(* PLC project contactor_1dir_2speed, Dassault Systèmes ControlBuild 2024x *)
(* stored: creationDateTime 2023-10-03T11:13:14-01:00 *)

(* This module simulates control system of motor. This motor has one direction and two speeds. This system is represented by two contactors. *)
FUNCTION_BLOCK equipment_library.contactor_1dir_2speed
  VAR_INPUT
    voltage380 : BOOL := true;
    cmdSupply : BOOL := true;
    sensorSupply : BOOL := true;
  END_VAR
  VAR_INPUT
    highSpeed : BOOL := false;
    lowSpeed : BOOL := false;
  END_VAR
  VAR_OUTPUT
    fwdHsState : BOOL := false;
    fwdLsState : BOOL := false;
  END_VAR
  VAR_OUTPUT
    highSpeedFB : BOOL := false;
    lowSpeedFB : BOOL := false;
    thermal : BOOL := false;
  END_VAR
  VAR
    memoHighSpeed : BOOL := false;
    memoLowSpeed : BOOL := false;
  END_VAR
  VAR CONSTANT
    highSpeedLogic : BOOL := true;
    lowSpeedLogic : BOOL := true;
    thermalLogic : BOOL := false;
  END_VAR
  VAR
    d_electrical : BOOL := false;
    v_d_electrical : BOOL := false;
    d_highSpeed : BOOL := false;
    v_d_highSpeed : BOOL := false;
    d_lowSpeed : BOOL := false;
    v_d_lowSpeed : BOOL := false;
  END_VAR


ACTION C_source_code:
/* ----------------------------------------------------------------	*/
/* Type : Model of Operative Behaviour					*/
/* Category :  Pre-actuators						*/
/* Author : Dassault Systemes						*/
/* Update date : June 2018							*/
/* ----------------------------------------------------------------	*/
/* This module simulates control system of motor. 			*/
/* This motor has one direction and two speeds. 			*/
/* This system is represented by two contactors. 			*/
/* It returns its state and sensors' feed-back.				*/
/* ----------------------------------------------------------------	*/

/* ----------------------------------------------------------------	*/
/* Management of orders from Control Part					*/
/*	if there is no power supply for command 				*/
/*         the contactor doesn't understand the control order		*/
/* Contactors are not mechanically bound					*/
/* ----------------------------------------------------------------	*/
memoLowSpeed = lowSpeed && !memoHighSpeed && cmdSupply && !d_electrical;
memoHighSpeed = highSpeed && !memoLowSpeed && cmdSupply && !d_electrical;


/* ----------------------------------------------------------------	*/
/* Calculation of the on-state of contactors				*/
/* ----------------------------------------------------------------	*/
fwdHsState=memoHighSpeed & voltage380;
fwdLsState=memoLowSpeed & voltage380;

/* ----------------------------------------------------------------	*/
/* Management of the thermal feed-back					*/
/* ----------------------------------------------------------------	*/
if (d_electrical) thermal=v_d_electrical;
else
	thermal= ! thermalLogic && sensorSupply;


/* ----------------------------------------------------------------	*/
/* Management of feedback to Control Part					*/
/*     if a fault is required, the contactor feed-back 		*/
/*		 takes a preset state.					*/
/*	if there is no power supply for sensor 				*/
/*         contactor feed-back returns nothing				*/
/*     else contactor feed-back returns the contactor state combined	*/
/*	    with wiring logic.						*/
/* ----------------------------------------------------------------	*/
if (d_highSpeed) highSpeedFB = v_d_highSpeed;
else 	
	highSpeedFB = (memoHighSpeed ^ ! highSpeedLogic) && sensorSupply;

if (d_lowSpeed) lowSpeedFB = v_d_lowSpeed;
else	
	lowSpeedFB = (memoLowSpeed ^ ! lowSpeedLogic) && sensorSupply;
END_ACTION
END_FUNCTION_BLOCK
